// TIA Portal V17 export
// export: Created 2025-11-26T18:31:36.4974107Z, ExportSetting WithDefaults, WithReadOnly, DisplayName Totally Integrated Automation Portal, DisplayVersion V17 Update 7, DisplayName TIA Portal Openness, DisplayVersion V17 Update 7, DisplayName TIA Portal Version Control Interface, DisplayVersion V17, DisplayName SINAMICS Startdrive Advanced, DisplayVersion V17 SP2, DisplayName SINAMICS Startdrive G110M, G120, G120C, G120D, G120P, G115D, DisplayVersion V17 SP2, DisplayName SINAMICS Startdrive G130, G150, S120, S150, SINAMICS MV, S210, DisplayVersion V17 SP2, DisplayName STEP 7 Professional, DisplayVersion V17 Update 7, DisplayName STEP 7 Safety, DisplayVersion V17 Update 6, DisplayName WinCC Advanced, DisplayVersion V17 Update 7, DisplayName SIMATIC Visualization Architect, DisplayVersion V17 Update 7
DATA_BLOCK "[nomeDB]"   // DB[numeroDB]
{ S7_Optimized_Access := 'TRUE' }
VERSION : 0.1
// DB= "11".DB?xxx.y
// stored: AutoNumber false, CodeModifiedDate 2024-09-18T07:15:12.2651526Z, CompileDate 2024-11-07T14:10:28.1057949Z, CreationDate 2024-05-14T09:07:19.2547822Z, DBAccessibleFromOPCUA true, DownloadWithoutReinit false, InterfaceModifiedDate 2024-10-18T13:52:06.5400932Z, IsConsistent true, IsKnowHowProtected false, IsOnlyStoredInLoadMemory false, IsPLCDB false, IsRetainMemResEnabled false, IsWriteProtectedInAS false, MemoryReserve 100, ModifiedDate 2024-10-18T13:52:06.5400932Z, ParameterModified 2024-09-18T07:15:12.2651526Z, StructureModified 2024-09-18T07:15:12.2651526Z
   VAR RETAIN
      Rob { ExternalAccessible := 'False'; ExternalVisible := 'False'; ExternalWritable := 'False'} : "ST_Rob";   // Roboter / Robot
      PG { ExternalAccessible := 'False'; ExternalVisible := 'False'; ExternalWritable := 'False'} : "ST_PG";   // Prozessgerätstruktur
      ExtMedienEIN { ExternalAccessible := 'False'; ExternalVisible := 'False'; ExternalWritable := 'False'} : Bool;   // externe Medien einschalten
      Warn { ExternalAccessible := 'False'; ExternalVisible := 'False'; ExternalWritable := 'False'} : Bool := false;   // Warnung / Varovanie
      Stoe { ExternalAccessible := 'False'; ExternalVisible := 'False'; ExternalWritable := 'False'} : Bool := false;   // Störung / Porucha
      Wart { ExternalAccessible := 'False'; ExternalVisible := 'False'; ExternalWritable := 'False'} : Bool := false;   // Wartung / Údržba
      PGWarn { ExternalAccessible := 'False'; ExternalVisible := 'False'; ExternalWritable := 'False'} : Bool := false;   // Warnung / Varovanie
      PGStoe { ExternalAccessible := 'False'; ExternalVisible := 'False'; ExternalWritable := 'False'} : Bool := false;   // Störung / Porucha
      PGWart { ExternalAccessible := 'False'; ExternalVisible := 'False'; ExternalWritable := 'False'} : Bool := false;   // Wartung / Údržba
      TZ { ExternalAccessible := 'False'; ExternalVisible := 'False'; ExternalWritable := 'False'} : "STB_Taktzeit_Plus";   // Taktzeit_Plus / Taktzeit Stopp Hifu
      FrgFolg1 { ExternalAccessible := 'False'; ExternalVisible := 'False'; ExternalWritable := 'False'} : Bool := false;   // Freigabe Folge 1 Schweissen 2-Tuerer
      FrgFolg2 { ExternalAccessible := 'False'; ExternalVisible := 'False'; ExternalWritable := 'False'} : Bool := false;   // Freigabe Folge 2 Schweissen 4-Tuerer
      FM { ExternalAccessible := 'False'; ExternalVisible := 'False'; ExternalWritable := 'False'} : Bool := false;   // Fertigmeldung Gesamt
      Frg_MaschSich { ExternalAccessible := 'False'; ExternalVisible := 'False'; ExternalWritable := 'False'} : Bool := false;   // Freigabe Maschinensicherheit Hifu
      StoeMedien { ExternalAccessible := 'False'; ExternalVisible := 'False'; ExternalWritable := 'False'} : Bool := false;   // Störung Roboter Medien
      PROFIe_Schlafmodus_aktiv { ExternalAccessible := 'False'; ExternalVisible := 'False'; ExternalWritable := 'False'} : Bool := false;   // PROFIenergy Schlafmodus aktiv
      PROFIe_FrgBedienung { ExternalAccessible := 'False'; ExternalVisible := 'False'; ExternalWritable := 'False'} : Bool := false;   // PROFIenergy Freigabe Bedienung
   END_VAR
BEGIN
END_DATA_BLOCK
